// Mitsubishi GX Works2 project: IOT_MES各功能   PLC: Q03UDV

PROGRAM #01
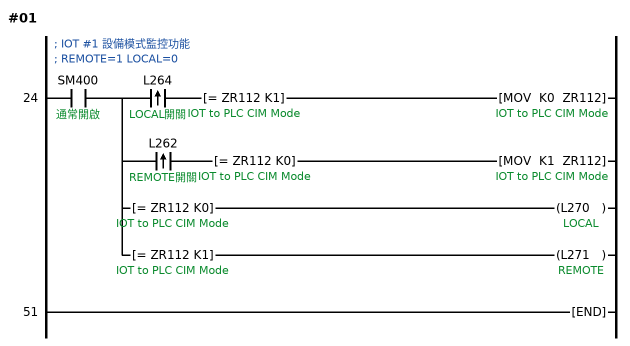
; IOT #1 設備模式監控功能
; REMOTE=1 LOCAL=0
24    LD      SM400  ; 通常開啟
      MPS
      ANDP    L264  ; LOCAL開關
      AND=    ZR112 K1  ; IOT to PLC CIM Mode
      MOV     K0 ZR112
      MRD
      ANDP    L262  ; REMOTE開關
      AND=    ZR112 K0  ; IOT to PLC CIM Mode
      MOV     K1 ZR112
      MRD
      AND=    ZR112 K0  ; IOT to PLC CIM Mode
      OUT     L270  ; LOCAL
      MPP
      AND=    ZR112 K1  ; IOT to PLC CIM Mode
      OUT     L271  ; REMOTE
51    END
END_PROGRAM

PROGRAM #02
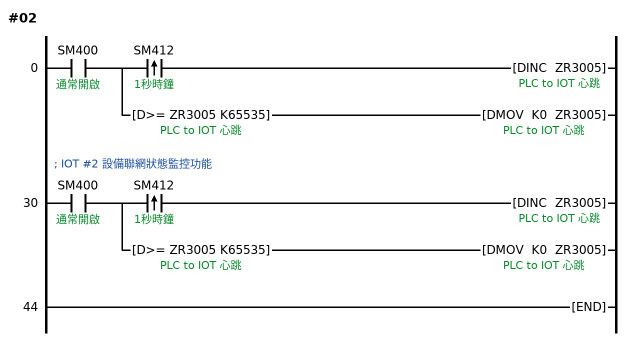
0     LD      SM400  ; 通常開啟
      MPS
      ANDP    SM412  ; 1秒時鐘
      DINC    ZR3005  ; PLC to IOT 心跳
      MPP
      ANDD>=  ZR3005 K65535  ; PLC to IOT 心跳
      DMOV    K0 ZR3005
; IOT #2 設備聯網狀態監控功能
30    LD      SM400  ; 通常開啟
      MPS
      ANDP    SM412  ; 1秒時鐘
      DINC    ZR3005
      MPP
      ANDD>=  ZR3005 K65535  ; PLC to IOT 心跳
      DMOV    K0 ZR3005
44    END
END_PROGRAM

PROGRAM #03
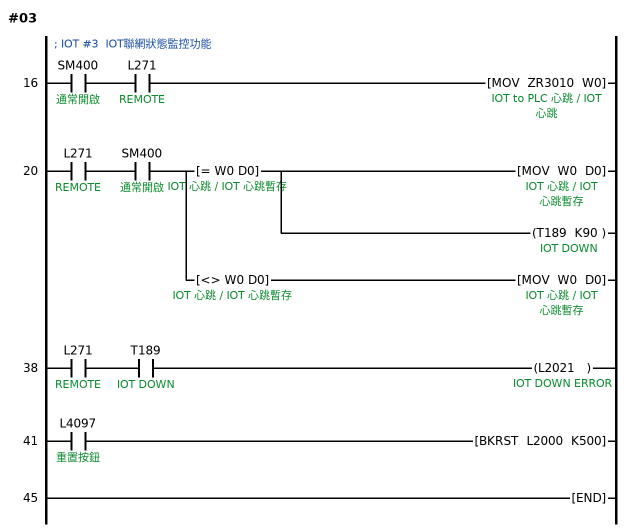
; IOT #3  IOT聯網狀態監控功能
16    LD      SM400  ; 通常開啟
      AND     L271  ; REMOTE
      MOV     ZR3010 W0  ; IOT to PLC 心跳 / IOT 心跳
20    LD      L271  ; REMOTE
      AND     SM400  ; 通常開啟
      MPS
      AND=    W0 D0  ; IOT 心跳 / IOT 心跳暫存
      MOV     W0 D0
      OUT     T189 K90  ; IOT DOWN
      MPP
      AND<>   W0 D0  ; IOT 心跳 / IOT 心跳暫存
      MOV     W0 D0
38    LD      L271  ; REMOTE
      AND     T189  ; IOT DOWN
      OUT     L2021  ; IOT DOWN ERROR
41    LD      L4097  ; 重置按鈕
      BKRST   L2000 K500
45    END
END_PROGRAM

PROGRAM #04
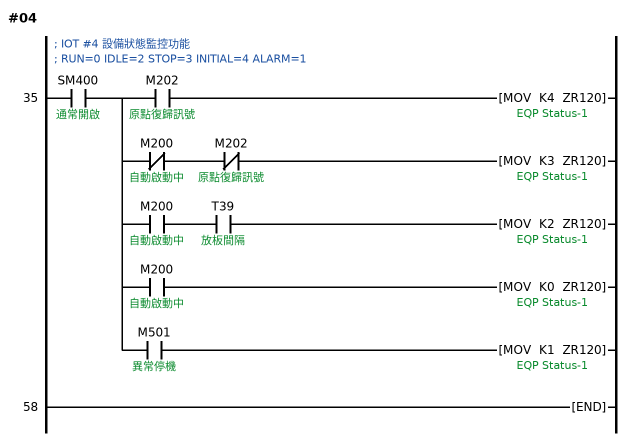
; IOT #4 設備狀態監控功能
; RUN=0 IDLE=2 STOP=3 INITIAL=4 ALARM=1
35    LD      SM400  ; 通常開啟
      MPS
      AND     M202  ; 原點復歸訊號
      MOV     K4 ZR120  ; EQP Status-1
      MRD
      ANI     M200  ; 自動啟動中
      ANI     M202  ; 原點復歸訊號
      MOV     K3 ZR120
      MRD
      AND     M200  ; 自動啟動中
      AND     T39  ; 放板間隔
      MOV     K2 ZR120
      MRD
      AND     M200  ; 自動啟動中
      MOV     K0 ZR120
      MPP
      AND     M501  ; 異常停機
      MOV     K1 ZR120
58    END
END_PROGRAM

PROGRAM #05
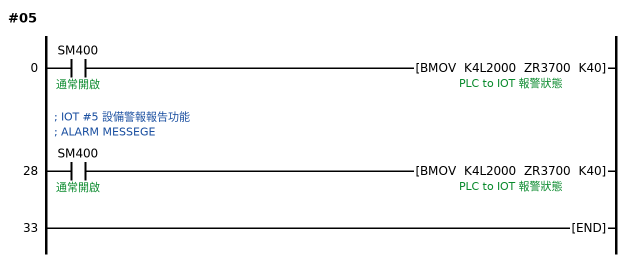
0     LD      SM400  ; 通常開啟
      BMOV    K4L2000 ZR3700 K40  ; PLC to IOT 報警狀態
; IOT #5 設備警報報告功能
; ALARM MESSEGE
28    LD      SM400  ; 通常開啟
      BMOV    K4L2000 ZR3700 K40
33    END
END_PROGRAM

PROGRAM #06
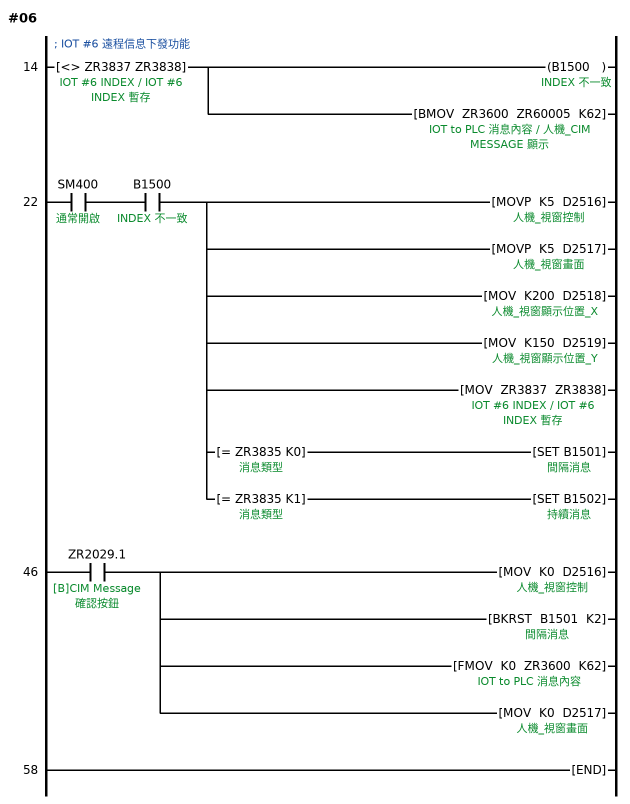
; IOT #6 遠程信息下發功能
14    LD<>    ZR3837 ZR3838  ; IOT #6 INDEX / IOT #6 INDEX 暫存
      OUT     B1500  ; INDEX 不一致
      BMOV    ZR3600 ZR60005 K62  ; IOT to PLC 消息內容 / 人機_CIM MESSAGE 顯示
22    LD      SM400  ; 通常開啟
      AND     B1500  ; INDEX 不一致
      MOVP    K5 D2516  ; 人機_視窗控制
      MOVP    K5 D2517  ; 人機_視窗畫面
      MOV     K200 D2518  ; 人機_視窗顯示位置_X
      MOV     K150 D2519  ; 人機_視窗顯示位置_Y
      MOV     ZR3837 ZR3838
      MPS
      AND=    ZR3835 K0  ; 消息類型
      SET     B1501  ; 間隔消息
      MPP
      AND=    ZR3835 K1  ; 消息類型
      SET     B1502  ; 持續消息
46    LD      ZR2029.1  ; [B]CIM Message 確認按鈕
      MOV     K0 D2516
      BKRST   B1501 K2
      FMOV    K0 ZR3600 K62
      MOV     K0 D2517
58    END
END_PROGRAM

PROGRAM #07
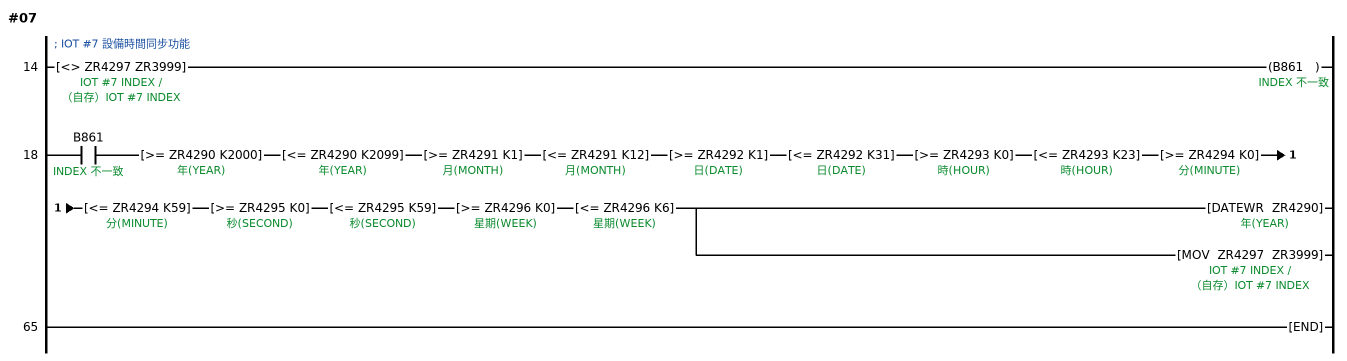
; IOT #7 設備時間同步功能
14    LD<>    ZR4297 ZR3999  ; IOT #7 INDEX / （自存）IOT #7 INDEX
      OUT     B861  ; INDEX 不一致
18    LD      B861  ; INDEX 不一致
      AND>=   ZR4290 K2000  ; 年(YEAR)
      AND<=   ZR4290 K2099  ; 年(YEAR)
      AND>=   ZR4291 K1  ; 月(MONTH)
      AND<=   ZR4291 K12  ; 月(MONTH)
      AND>=   ZR4292 K1  ; 日(DATE)
      AND<=   ZR4292 K31  ; 日(DATE)
      AND>=   ZR4293 K0  ; 時(HOUR)
      AND<=   ZR4293 K23  ; 時(HOUR)
      AND>=   ZR4294 K0  ; 分(MINUTE)
      AND<=   ZR4294 K59  ; 分(MINUTE)
      AND>=   ZR4295 K0  ; 秒(SECOND)
      AND<=   ZR4295 K59  ; 秒(SECOND)
      AND>=   ZR4296 K0  ; 星期(WEEK)
      AND<=   ZR4296 K6  ; 星期(WEEK)
      DATEWR  ZR4290
      MOV     ZR4297 ZR3999
65    END
END_PROGRAM

PROGRAM #09
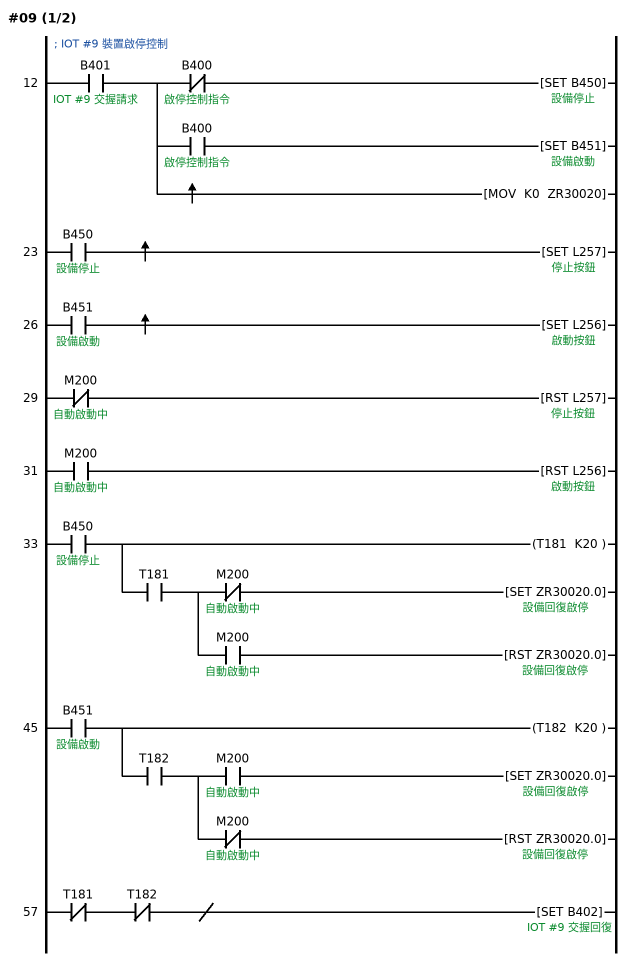
; IOT #9 裝置啟停控制
12    LD      B401  ; IOT #9 交握請求
      MPS
      ANI     B400  ; 啟停控制指令
      SET     B450  ; 設備停止
      MRD
      AND     B400  ; 啟停控制指令
      SET     B451  ; 設備啟動
      MPP
      MEP
      MOV     K0 ZR30020
23    LD      B450  ; 設備停止
      MEP
      SET     L257  ; 停止按鈕
26    LD      B451  ; 設備啟動
      MEP
      SET     L256  ; 啟動按鈕
29    LDI     M200  ; 自動啟動中
      RST     L257  ; 停止按鈕
31    LD      M200  ; 自動啟動中
      RST     L256  ; 啟動按鈕
33    LD      B450  ; 設備停止
      OUT     T181 K20
      AND     T181
      MPS
      ANI     M200  ; 自動啟動中
      SET     ZR30020.0  ; 設備回復啟停
      MPP
      AND     M200  ; 自動啟動中
      RST     ZR30020.0  ; 設備回復啟停
45    LD      B451  ; 設備啟動
      OUT     T182 K20
      AND     T182
      MPS
      AND     M200  ; 自動啟動中
      SET     ZR30020.0  ; 設備回復啟停
      MPP
      ANI     M200  ; 自動啟動中
      RST     ZR30020.0  ; 設備回復啟停
57    LDI     T181
      ANI     T182
      INV
      SET     B402  ; IOT #9 交握回復
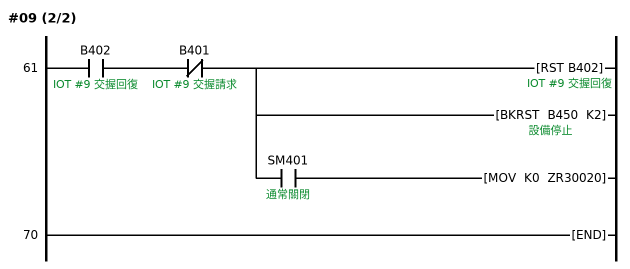
61    LD      B402  ; IOT #9 交握回復
      ANI     B401  ; IOT #9 交握請求
      RST     B402  ; IOT #9 交握回復
      BKRST   B450 K2
      AND     SM401  ; 通常關閉
      MOV     K0 ZR30020
70    END
END_PROGRAM

PROGRAM #10
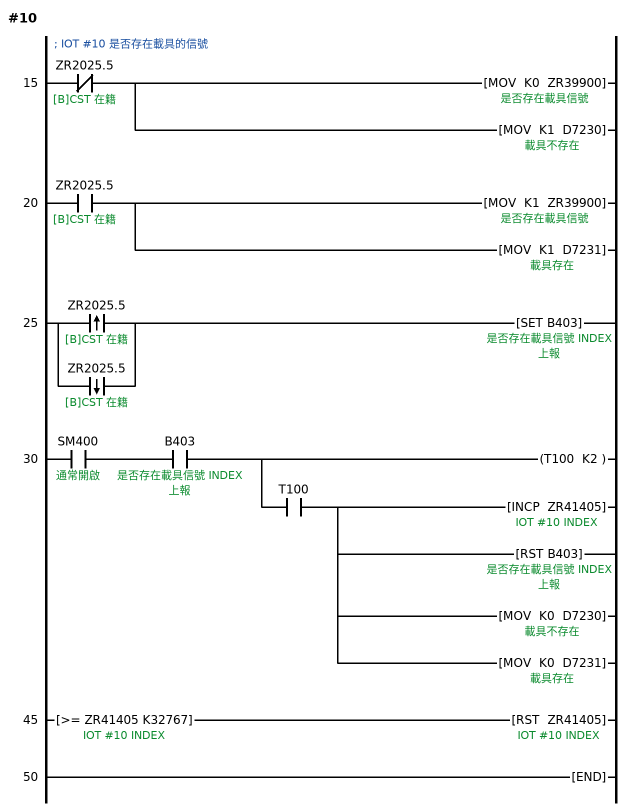
; IOT #10 是否存在載具的信號
15    LDI     ZR2025.5  ; [B]CST 在籍
      MOV     K0 ZR39900  ; 是否存在載具信號
      MOV     K1 D7230  ; 載具不存在
20    LD      ZR2025.5  ; [B]CST 在籍
      MOV     K1 ZR39900
      MOV     K1 D7231  ; 載具存在
25    LDP     ZR2025.5  ; [B]CST 在籍
      ORF     ZR2025.5  ; [B]CST 在籍
      SET     B403  ; 是否存在載具信號 INDEX 上報
30    LD      SM400  ; 通常開啟
      AND     B403  ; 是否存在載具信號 INDEX 上報
      OUT     T100 K2
      AND     T100
      INCP    ZR41405  ; IOT #10 INDEX
      RST     B403  ; 是否存在載具信號 INDEX 上報
      MOV     K0 D7230
      MOV     K0 D7231
45    LD>=    ZR41405 K32767  ; IOT #10 INDEX
      RST     ZR41405  ; IOT #10 INDEX
50    END
END_PROGRAM

PROGRAM #11
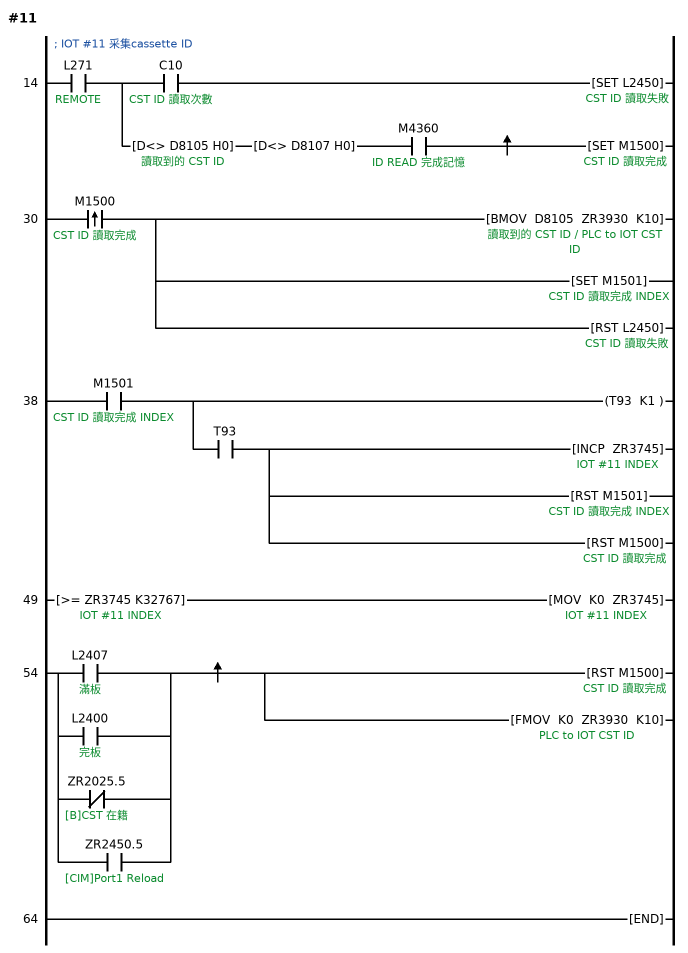
; IOT #11 采集cassette ID
14    LD      L271  ; REMOTE
      MPS
      AND     C10  ; CST ID 讀取次數
      SET     L2450  ; CST ID 讀取失敗
      MPP
      ANDD<>  D8105 H0  ; 讀取到的 CST ID
      ANDD<>  D8107 H0
      AND     M4360  ; ID READ 完成記憶
      MEP
      SET     M1500  ; CST ID 讀取完成
30    LDP     M1500  ; CST ID 讀取完成
      BMOV    D8105 ZR3930 K10  ; PLC to IOT CST ID
      SET     M1501  ; CST ID 讀取完成 INDEX
      RST     L2450  ; CST ID 讀取失敗
38    LD      M1501  ; CST ID 讀取完成 INDEX
      OUT     T93 K1
      AND     T93
      INCP    ZR3745  ; IOT #11 INDEX
      RST     M1501  ; CST ID 讀取完成 INDEX
      RST     M1500  ; CST ID 讀取完成
49    LD>=    ZR3745 K32767  ; IOT #11 INDEX
      MOV     K0 ZR3745
54    LD      L2407  ; 滿板
      OR      L2400  ; 完板
      ORI     ZR2025.5  ; [B]CST 在籍
      OR      ZR2450.5  ; [CIM]Port1 Reload
      MEP
      RST     M1500  ; CST ID 讀取完成
      FMOV    K0 ZR3930 K10
64    END
END_PROGRAM

PROGRAM 收#12#13
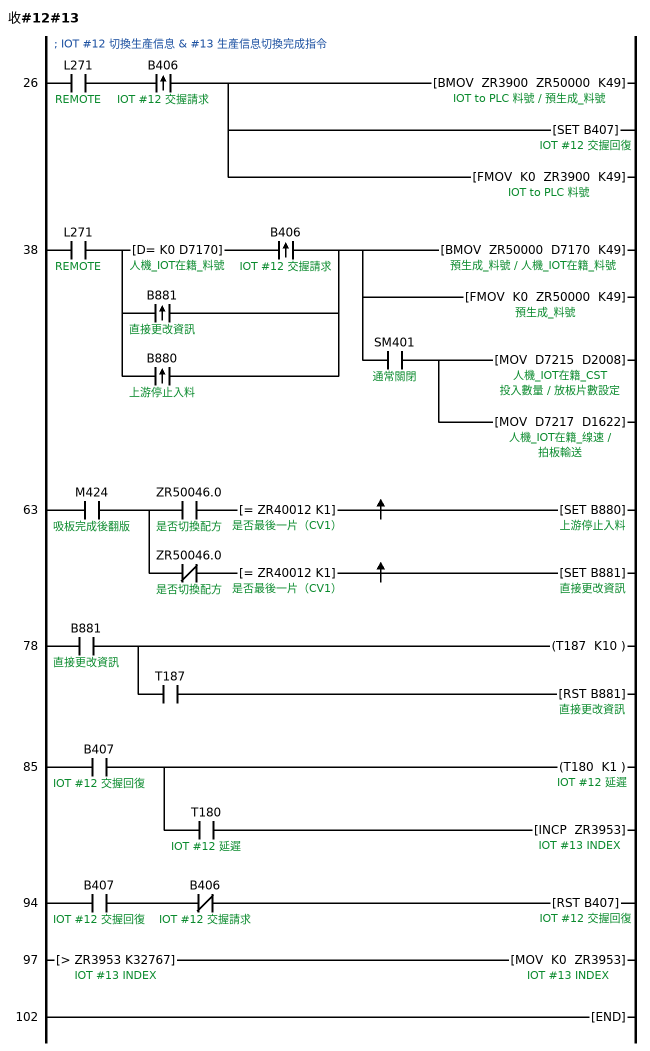
; IOT #12 切換生產信息 & #13 生產信息切換完成指令
26    LD      L271  ; REMOTE
      ANDP    B406  ; IOT #12 交握請求
      BMOV    ZR3900 ZR50000 K49  ; IOT to PLC 料號 / 預生成_料號
      SET     B407  ; IOT #12 交握回復
      FMOV    K0 ZR3900 K49
38    LD      L271  ; REMOTE
      LDD=    K0 D7170  ; 人機_IOT在籍_料號
      ANDP    B406  ; IOT #12 交握請求
      ORP     B881  ; 直接更改資訊
      ORP     B880  ; 上游停止入料
      ANB
      BMOV    ZR50000 D7170 K49
      FMOV    K0 ZR50000 K49
      AND     SM401  ; 通常關閉
      MOV     D7215 D2008  ; 人機_IOT在籍_CST 投入數量 / 放板片數設定
      MOV     D7217 D1622  ; 人機_IOT在籍_缐速 / 拍板輸送
63    LD      M424  ; 吸板完成後翻版
      MPS
      AND     ZR50046.0  ; 是否切換配方
      AND=    ZR40012 K1  ; 是否最後一片（CV1）
      MEP
      SET     B880  ; 上游停止入料
      MPP
      ANI     ZR50046.0  ; 是否切換配方
      AND=    ZR40012 K1  ; 是否最後一片（CV1）
      MEP
      SET     B881  ; 直接更改資訊
78    LD      B881  ; 直接更改資訊
      OUT     T187 K10
      AND     T187
      RST     B881  ; 直接更改資訊
85    LD      B407  ; IOT #12 交握回復
      OUT     T180 K1  ; IOT #12 延遲
      AND     T180  ; IOT #12 延遲
      INCP    ZR3953  ; IOT #13 INDEX
94    LD      B407  ; IOT #12 交握回復
      ANI     B406  ; IOT #12 交握請求
      RST     B407  ; IOT #12 交握回復
97    LD>     ZR3953 K32767  ; IOT #13 INDEX
      MOV     K0 ZR3953
102   END
END_PROGRAM

PROGRAM 收#14
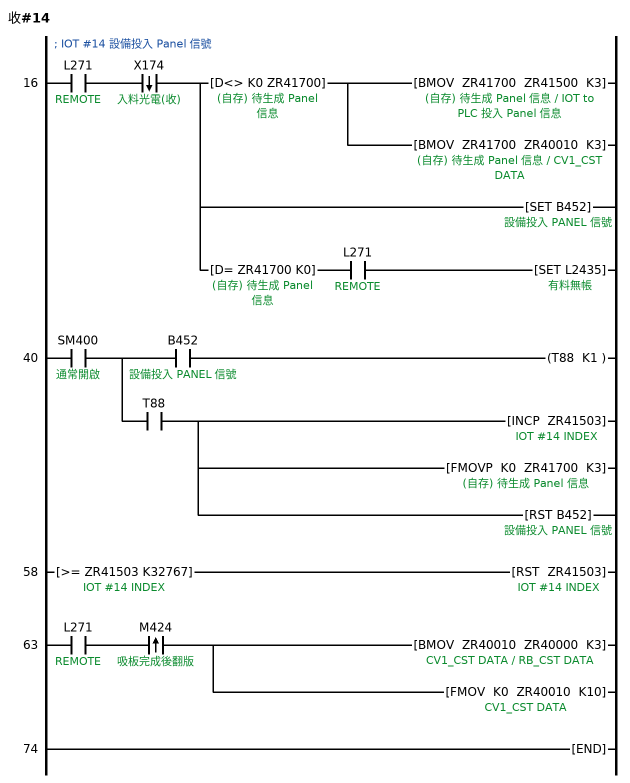
; IOT #14 設備投入 Panel 信號
16    LD      L271  ; REMOTE
      ANDF    X174  ; 入料光電(收)
      MPS
      ANDD<>  K0 ZR41700  ; (自存) 待生成 Panel 信息
      BMOV    ZR41700 ZR41500 K3  ; IOT to PLC 投入 Panel 信息
      BMOV    ZR41700 ZR40010 K3  ; CV1_CST DATA
      MPP
      SET     B452  ; 設備投入 PANEL 信號
      ANDD=   ZR41700 K0  ; (自存) 待生成 Panel 信息
      AND     L271  ; REMOTE
      SET     L2435  ; 有料無帳
40    LD      SM400  ; 通常開啟
      MPS
      AND     B452  ; 設備投入 PANEL 信號
      OUT     T88 K1
      MPP
      AND     T88
      INCP    ZR41503  ; IOT #14 INDEX
      FMOVP   K0 ZR41700 K3
      RST     B452  ; 設備投入 PANEL 信號
58    LD>=    ZR41503 K32767  ; IOT #14 INDEX
      RST     ZR41503  ; IOT #14 INDEX
63    LD      L271  ; REMOTE
      ANDP    M424  ; 吸板完成後翻版
      BMOV    ZR40010 ZR40000 K3  ; RB_CST DATA
      FMOV    K0 ZR40010 K10
74    END
END_PROGRAM

PROGRAM 收#15
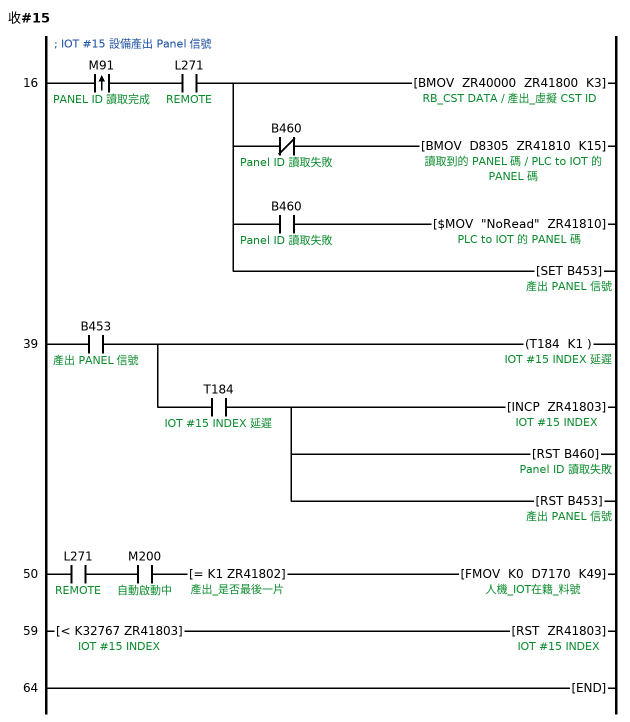
; IOT #15 設備產出 Panel 信號
16    LDP     M91  ; PANEL ID 讀取完成
      AND     L271  ; REMOTE
      BMOV    ZR40000 ZR41800 K3  ; RB_CST DATA / 產出_虛擬 CST ID
      MPS
      ANI     B460  ; Panel ID 讀取失敗
      BMOV    D8305 ZR41810 K15  ; 讀取到的 PANEL 碼 / PLC to IOT 的 PANEL 碼
      MRD
      AND     B460  ; Panel ID 讀取失敗
      $MOV    "NoRead" ZR41810
      MPP
      SET     B453  ; 產出 PANEL 信號
39    LD      B453  ; 產出 PANEL 信號
      OUT     T184 K1  ; IOT #15 INDEX 延遲
      AND     T184  ; IOT #15 INDEX 延遲
      INCP    ZR41803  ; IOT #15 INDEX
      RST     B460  ; Panel ID 讀取失敗
      RST     B453  ; 產出 PANEL 信號
50    LD      L271  ; REMOTE
      AND     M200  ; 自動啟動中
      AND=    K1 ZR41802  ; 產出_是否最後一片
      FMOV    K0 D7170 K49  ; 人機_IOT在籍_料號
59    LD<     K32767 ZR41803  ; IOT #15 INDEX
      RST     ZR41803  ; IOT #15 INDEX
64    END
END_PROGRAM

PROGRAM #16
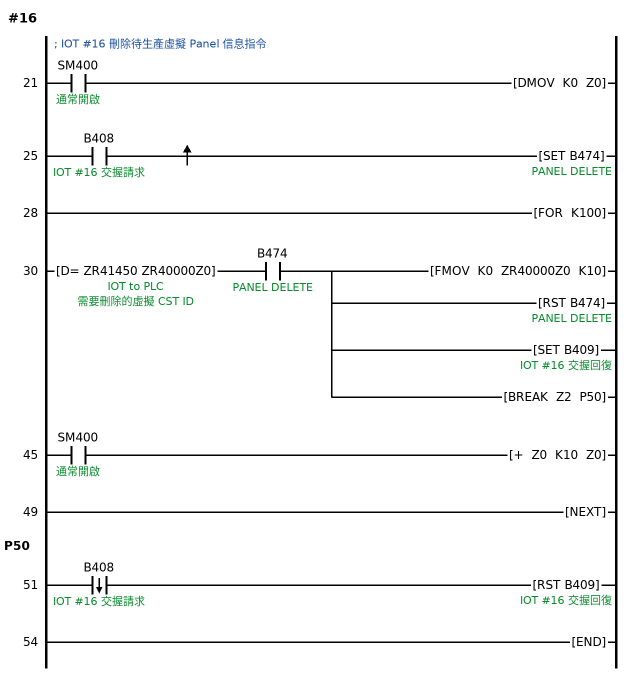
; IOT #16 刪除待生產虛擬 Panel 信息指令
21    LD      SM400  ; 通常開啟
      DMOV    K0 Z0
25    LD      B408  ; IOT #16 交握請求
      MEP
      SET     B474  ; PANEL DELETE
28    FOR     K100
30    LDD=    ZR41450 ZR40000Z0  ; IOT to PLC 需要刪除的虛擬 CST ID
      AND     B474  ; PANEL DELETE
      FMOV    K0 ZR40000Z0 K10
      RST     B474  ; PANEL DELETE
      SET     B409  ; IOT #16 交握回復
      BREAK   Z2 P50
45    LD      SM400  ; 通常開啟
      +       Z0 K10 Z0
49    NEXT
      P50
51    LDF     B408  ; IOT #16 交握請求
      RST     B409  ; IOT #16 交握回復
54    END
END_PROGRAM

PROGRAM 收#17
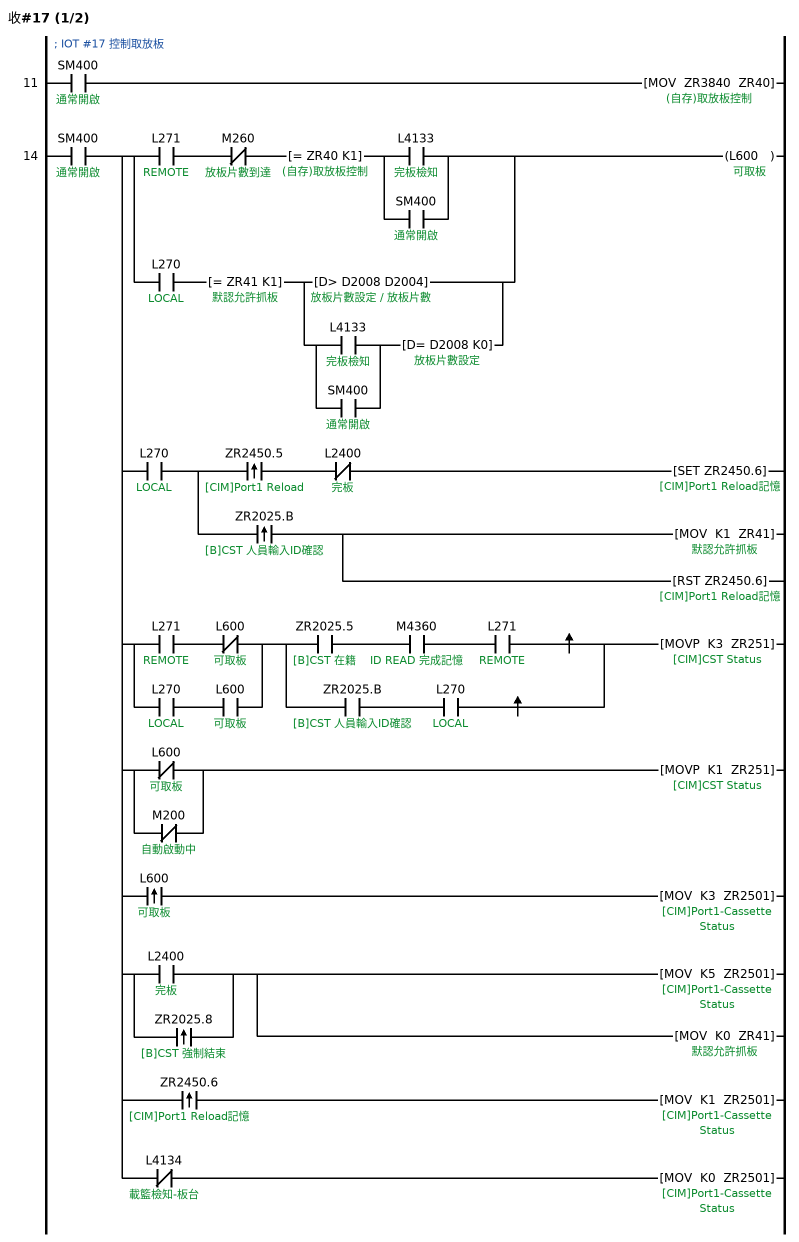
; IOT #17 控制取放板
11    LD      SM400  ; 通常開啟
      MOV     ZR3840 ZR40  ; (自存)取放板控制
14    LD      SM400  ; 通常開啟
      MPS
      LD      L271  ; REMOTE
      ANI     M260  ; 放板片數到達
      AND=    ZR40 K1  ; (自存)取放板控制
      LD      L4133  ; 完板檢知
      OR      SM400  ; 通常開啟
      ANB
      LD      L270  ; LOCAL
      AND=    ZR41 K1  ; 默認允許抓板
      LDD>    D2008 D2004  ; 放板片數設定 / 放板片數
      LD      L4133  ; 完板檢知
      OR      SM400  ; 通常開啟
      ANDD=   D2008 K0  ; 放板片數設定
      ORB
      ANB
      ORB
      ANB
      OUT     L600  ; 可取板
      MRD
      AND     L270  ; LOCAL
      MPS
      ANDP    ZR2450.5  ; [CIM]Port1 Reload
      ANI     L2400  ; 完板
      SET     ZR2450.6  ; [CIM]Port1 Reload記憶
      MPP
      ANDP    ZR2025.B  ; [B]CST 人員輸入ID確認
      MOV     K1 ZR41
      RST     ZR2450.6  ; [CIM]Port1 Reload記憶
      MRD
      LD      L271  ; REMOTE
      ANI     L600  ; 可取板
      LD      L270  ; LOCAL
      AND     L600  ; 可取板
      ORB
      ANB
      LD      ZR2025.5  ; [B]CST 在籍
      AND     M4360  ; ID READ 完成記憶
      AND     L271  ; REMOTE
      MEP
      LD      ZR2025.B  ; [B]CST 人員輸入ID確認
      AND     L270  ; LOCAL
      MEP
      ORB
      ANB
      MOVP    K3 ZR251  ; [CIM]CST Status
      MRD
      LDI     L600  ; 可取板
      ORI     M200  ; 自動啟動中
      ANB
      MOVP    K1 ZR251
      MRD
      ANDP    L600  ; 可取板
      MOV     K3 ZR2501  ; [CIM]Port1-Cassette Status
      MRD
      LD      L2400  ; 完板
      ORP     ZR2025.8  ; [B]CST 強制結束
      ANB
      MOV     K5 ZR2501
      MOV     K0 ZR41
      MRD
      ANDP    ZR2450.6  ; [CIM]Port1 Reload記憶
      MOV     K1 ZR2501
      MPP
      ANI     L4134  ; 載籃檢知-板台
      MOV     K0 ZR2501
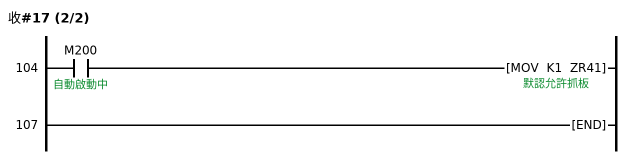
104   LD      M200  ; 自動啟動中
      MOV     K1 ZR41
107   END
END_PROGRAM

PROGRAM #19
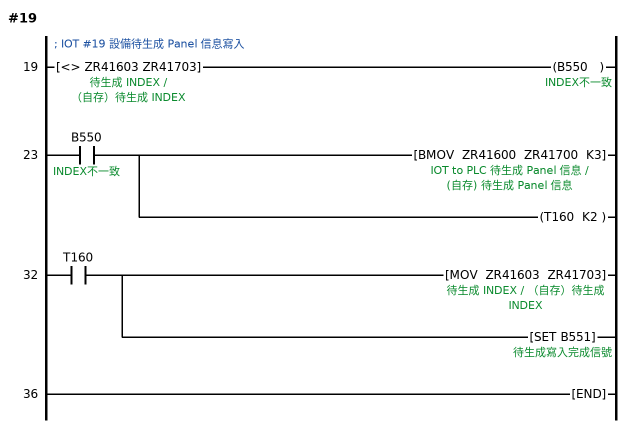
; IOT #19 設備待生成 Panel 信息寫入
19    LD<>    ZR41603 ZR41703  ; 待生成 INDEX / （自存）待生成 INDEX
      OUT     B550  ; INDEX不一致
23    LD      B550  ; INDEX不一致
      BMOV    ZR41600 ZR41700 K3  ; IOT to PLC 待生成 Panel 信息 / (自存) 待生成 Panel 信息
      OUT     T160 K2
32    LD      T160
      MOV     ZR41603 ZR41703
      SET     B551  ; 待生成寫入完成信號
36    END
END_PROGRAM

PROGRAM #20
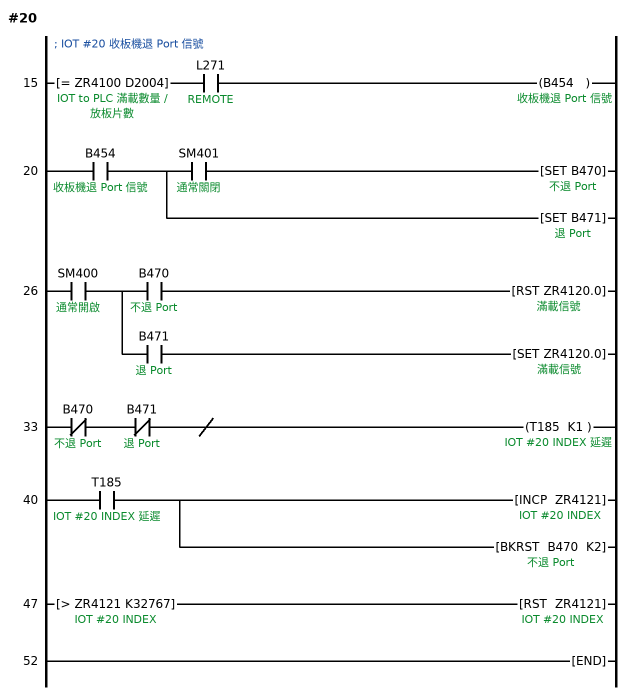
; IOT #20 收板機退 Port 信號
15    LD=     ZR4100 D2004  ; IOT to PLC 滿載數量 / 放板片數
      AND     L271  ; REMOTE
      OUT     B454  ; 收板機退 Port 信號
20    LD      B454  ; 收板機退 Port 信號
      MPS
      AND     SM401  ; 通常關閉
      SET     B470  ; 不退 Port
      MPP
      SET     B471  ; 退 Port
26    LD      SM400  ; 通常開啟
      MPS
      AND     B470  ; 不退 Port
      RST     ZR4120.0  ; 滿載信號
      MPP
      AND     B471  ; 退 Port
      SET     ZR4120.0  ; 滿載信號
33    LDI     B470  ; 不退 Port
      ANI     B471  ; 退 Port
      INV
      OUT     T185 K1  ; IOT #20 INDEX 延遲
40    LD      T185  ; IOT #20 INDEX 延遲
      INCP    ZR4121  ; IOT #20 INDEX
      BKRST   B470 K2
47    LD>     ZR4121 K32767  ; IOT #20 INDEX
      RST     ZR4121  ; IOT #20 INDEX
52    END
END_PROGRAM

PROGRAM #21
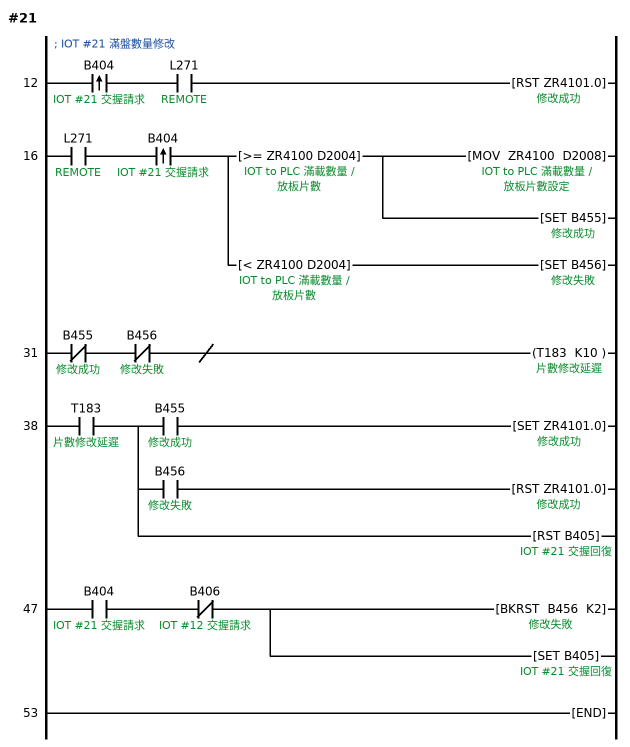
; IOT #21 滿盤數量修改
12    LDP     B404  ; IOT #21 交握請求
      AND     L271  ; REMOTE
      RST     ZR4101.0  ; 修改成功
16    LD      L271  ; REMOTE
      ANDP    B404  ; IOT #21 交握請求
      MPS
      AND>=   ZR4100 D2004  ; IOT to PLC 滿載數量 / 放板片數
      MOV     ZR4100 D2008  ; 放板片數設定
      SET     B455  ; 修改成功
      MPP
      AND<    ZR4100 D2004  ; IOT to PLC 滿載數量 / 放板片數
      SET     B456  ; 修改失敗
31    LDI     B455  ; 修改成功
      ANI     B456  ; 修改失敗
      INV
      OUT     T183 K10  ; 片數修改延遲
38    LD      T183  ; 片數修改延遲
      MPS
      AND     B455  ; 修改成功
      SET     ZR4101.0  ; 修改成功
      MRD
      AND     B456  ; 修改失敗
      RST     ZR4101.0  ; 修改成功
      MPP
      RST     B405  ; IOT #21 交握回復
47    LD      B404  ; IOT #21 交握請求
      ANI     B406  ; IOT #12 交握請求
      BKRST   B456 K2
      SET     B405  ; IOT #21 交握回復
53    END
END_PROGRAM

PROGRAM 放#12#13
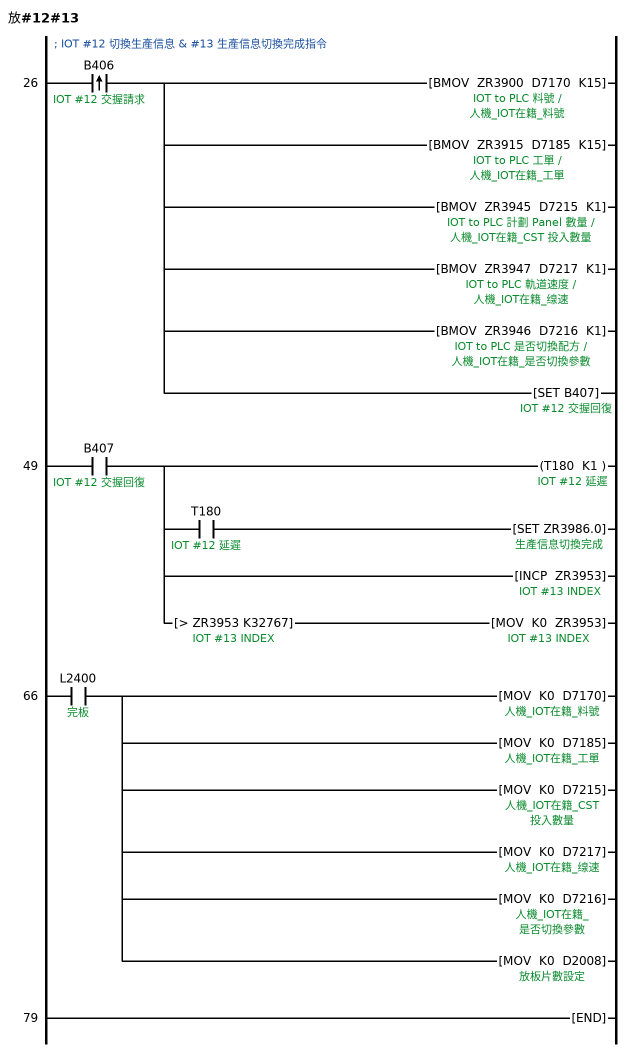
; IOT #12 切換生產信息 & #13 生產信息切換完成指令
26    LDP     B406  ; IOT #12 交握請求
      BMOV    ZR3900 D7170 K15  ; IOT to PLC 料號 / 人機_IOT在籍_料號
      BMOV    ZR3915 D7185 K15  ; IOT to PLC 工單 / 人機_IOT在籍_工單
      BMOV    ZR3945 D7215 K1  ; IOT to PLC 計劃 Panel 數量 / 人機_IOT在籍_CST 投入數量
      BMOV    ZR3947 D7217 K1  ; IOT to PLC 軌道速度 / 人機_IOT在籍_缐速
      BMOV    ZR3946 D7216 K1  ; IOT to PLC 是否切換配方 / 人機_IOT在籍_是否切換參數
      SET     B407  ; IOT #12 交握回復
49    LD      B407  ; IOT #12 交握回復
      OUT     T180 K1  ; IOT #12 延遲
      MPS
      AND     T180  ; IOT #12 延遲
      SET     ZR3986.0  ; 生產信息切換完成
      MPP
      INCP    ZR3953  ; IOT #13 INDEX
      AND>    ZR3953 K32767  ; IOT #13 INDEX
      MOV     K0 ZR3953
66    LD      L2400  ; 完板
      MOV     K0 D7170
      MOV     K0 D7185
      MOV     K0 D7215
      MOV     K0 D7217
      MOV     K0 D7216
      MOV     K0 D2008  ; 放板片數設定
79    END
END_PROGRAM

PROGRAM 放#14
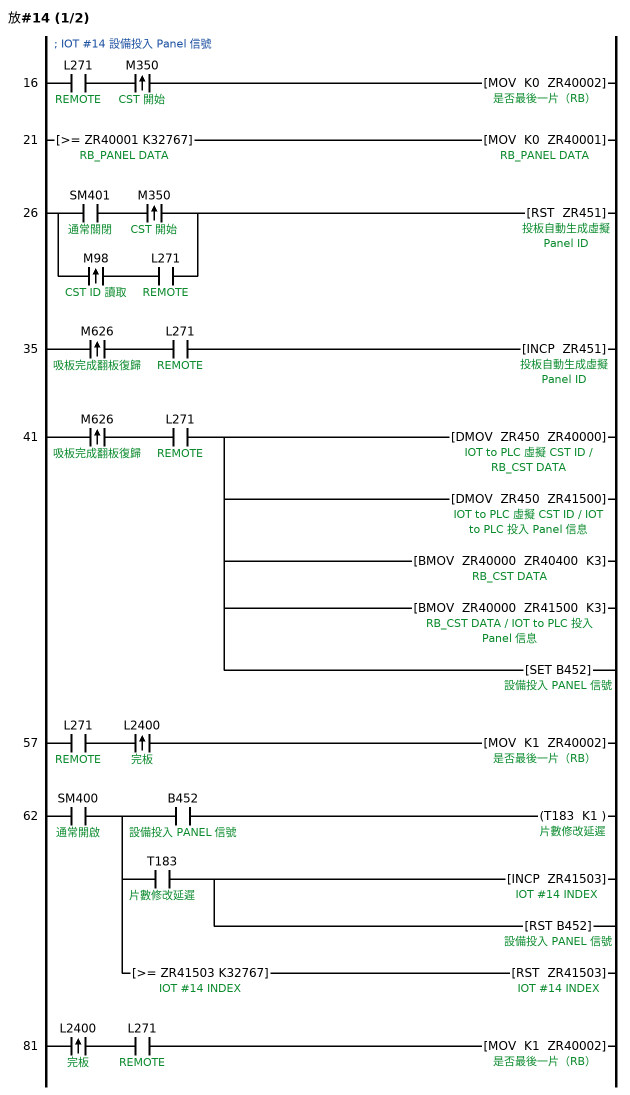
; IOT #14 設備投入 Panel 信號
16    LD      L271  ; REMOTE
      ANDP    M350  ; CST 開始
      MOV     K0 ZR40002  ; 是否最後一片（RB）
21    LD>=    ZR40001 K32767  ; RB_PANEL DATA
      MOV     K0 ZR40001
26    LD      SM401  ; 通常關閉
      ANDP    M350  ; CST 開始
      LDP     M98  ; CST ID 讀取
      AND     L271  ; REMOTE
      ORB
      RST     ZR451  ; 投板自動生成虛擬 Panel ID
35    LDP     M626  ; 吸板完成翻板復歸
      AND     L271  ; REMOTE
      INCP    ZR451
41    LDP     M626  ; 吸板完成翻板復歸
      AND     L271  ; REMOTE
      DMOV    ZR450 ZR40000  ; IOT to PLC 虛擬 CST ID / RB_CST DATA
      DMOV    ZR450 ZR41500  ; IOT to PLC 投入 Panel 信息
      BMOV    ZR40000 ZR40400 K3
      BMOV    ZR40000 ZR41500 K3
      SET     B452  ; 設備投入 PANEL 信號
57    LD      L271  ; REMOTE
      ANDP    L2400  ; 完板
      MOV     K1 ZR40002
62    LD      SM400  ; 通常開啟
      MPS
      AND     B452  ; 設備投入 PANEL 信號
      OUT     T183 K1  ; 片數修改延遲
      MRD
      AND     T183  ; 片數修改延遲
      INCP    ZR41503  ; IOT #14 INDEX
      RST     B452  ; 設備投入 PANEL 信號
      MPP
      AND>=   ZR41503 K32767  ; IOT #14 INDEX
      RST     ZR41503  ; IOT #14 INDEX
81    LDP     L2400  ; 完板
      AND     L271  ; REMOTE
      MOV     K1 ZR40002
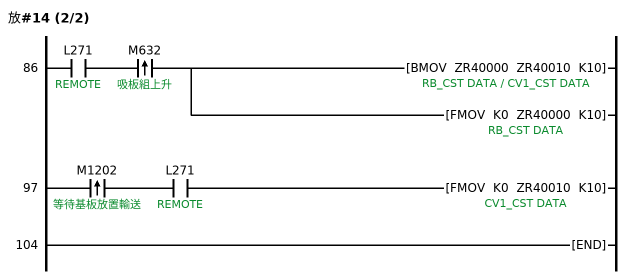
86    LD      L271  ; REMOTE
      ANDP    M632  ; 吸板組上升
      BMOV    ZR40000 ZR40010 K10  ; CV1_CST DATA
      FMOV    K0 ZR40000 K10
97    LDP     M1202  ; 等待基板放置輸送
      AND     L271  ; REMOTE
      FMOV    K0 ZR40010 K10
104   END
END_PROGRAM

PROGRAM 放#15
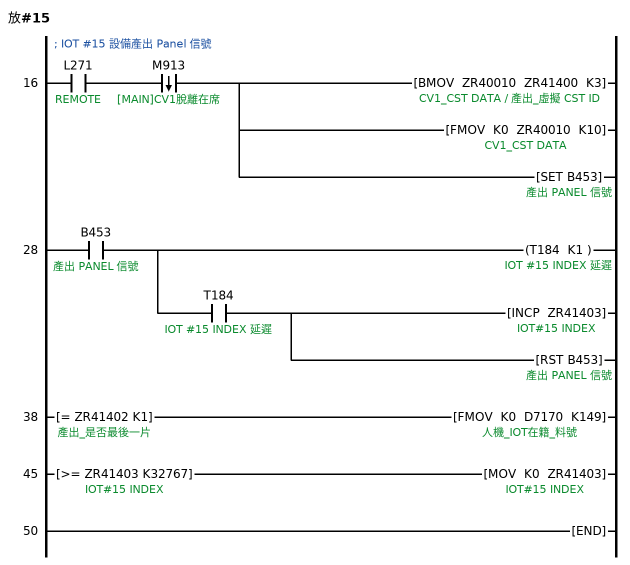
; IOT #15 設備產出 Panel 信號
16    LD      L271  ; REMOTE
      ANDF    M913  ; [MAIN]CV1脫離在席
      BMOV    ZR40010 ZR41400 K3  ; CV1_CST DATA / 產出_虛擬 CST ID
      FMOV    K0 ZR40010 K10
      SET     B453  ; 產出 PANEL 信號
28    LD      B453  ; 產出 PANEL 信號
      OUT     T184 K1  ; IOT #15 INDEX 延遲
      AND     T184  ; IOT #15 INDEX 延遲
      INCP    ZR41403  ; IOT#15 INDEX
      RST     B453  ; 產出 PANEL 信號
38    LD=     ZR41402 K1  ; 產出_是否最後一片
      FMOV    K0 D7170 K149  ; 人機_IOT在籍_料號
45    LD>=    ZR41403 K32767  ; IOT#15 INDEX
      MOV     K0 ZR41403
50    END
END_PROGRAM

PROGRAM 放#17
